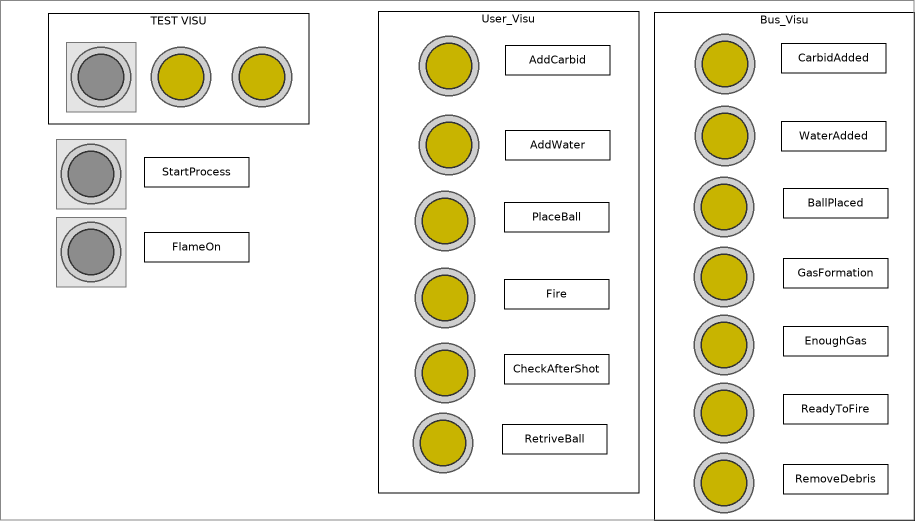
VISUALIZATION Visualization_Carbid_V2  // 915x521
    Rectangle (378,11 261x482), "User_Visu"
    Rectangle (48,13 261x111), "TEST VISU"
    Lamp1 (146,42 70x70), variable: Lamp, style: Lamp-Lamp1-Yellow
    PushSwitch (66,42 70x70), variable: Button, behaviour: TAP, style: Switch-PushSwitch-Gray
    Lamp1 (227,42 70x70), variable: BlinkingLamp, style: Lamp-Lamp1-Yellow
    PushSwitchLed (56,139 70x70), variable: StartProcess, behaviour: TOGGLE, style: Switch-PushSwitchLed-Gray
    PushSwitch (56,217 70x70), variable: FlameOn, behaviour: TAP, style: Switch-PushSwitch-Gray
    Rectangle (144,157 105x30), "StartProcess"
    Rectangle (144,232 105x30), "FlameOn"
    Lamp1 (414,31 70x70), variable: AddCarbid, style: Lamp-Lamp1-Yellow
    Lamp1 (414,110 70x70), variable: AddWater, style: Lamp-Lamp1-Yellow
    Rectangle (505,45 105x30), "AddCarbid"
    Rectangle (505,130 105x30), "AddWater"
    Lamp1 (410,186 70x70), variable: PlaceBall, style: Lamp-Lamp1-Yellow
    Rectangle (504,202 105x30), "PlaceBall"
    Lamp1 (410,263 70x70), variable: Fire, style: Lamp-Lamp1-Yellow
    Rectangle (504,279 105x30), "Fire"
    Lamp1 (410,338 70x70), variable: CheckAfterShot, style: Lamp-Lamp1-Yellow
    Rectangle (504,354 105x30), "CheckAfterShot"
    Rectangle (654,12 261x509), "Bus_Visu"
    Lamp1 (690,29 70x70), variable: CarbidAdded, style: Lamp-Lamp1-Yellow
    Lamp1 (690,101 70x70), variable: WaterAdded, style: Lamp-Lamp1-Yellow
    Rectangle (781,43 105x30), "CarbidAdded"
    Rectangle (781,121 105x30), "WaterAdded"
    Lamp1 (689,242 70x70), variable: GasFormation, style: Lamp-Lamp1-Yellow
    Rectangle (783,258 105x30), "GasFormation"
    Lamp1 (689,310 70x70), variable: EnoughGas, style: Lamp-Lamp1-Yellow
    Rectangle (783,326 105x30), "EnoughGas"
    Lamp1 (689,378 70x70), variable: ReadyToFire, style: Lamp-Lamp1-Yellow
    Rectangle (783,394 105x30), "ReadyToFire"
    Lamp1 (408,408 70x70), variable: RetrieveBall, style: Lamp-Lamp1-Yellow
    Rectangle (502,424 105x30), "RetriveBall"
    Lamp1 (689,448 70x70), variable: RemoveDebris, style: Lamp-Lamp1-Yellow
    Rectangle (783,464 105x30), "RemoveDebris"
    Lamp1 (689,172 70x70), variable: BallPlaced, style: Lamp-Lamp1-Yellow
    Rectangle (783,188 105x30), "BallPlaced"
END_VISUALIZATION

(* stored: Version 1.1.0.1, ProductVersion 3.1.4024.12
   Visu Visualization_Carbid_V2: Id {e94723d5-68cf-4fff-ae03-6c44a1cb2a05} *)
